{attribute 'GeneratedUsingTerminal: IODEVICETYPE_ETHERCATPROT'}
{attribute addProperty BoxType "IODEVICETYPE_ETHERCATPROT"}
{attribute addProperty Id "Beckhoff_BKxxxxBeckhoff_BKxxxx_735133AB0Beckhoff_CUxxxxBeckhoff_CUxxxx_E18DC8DB94Beckhoff_CXxxxxBeckhoff_CXxxxx_C55F0A74176TcTerminals210_EK1100_1TcTerminals210_EK1100_1_5C7783790TcTerminals210_EK1100_2TcTerminals210_EK1100_2_50C143310SyncUnitsSyncUnits_99E584AF18InputsInputs_25A0042B160OutputsOutputs_2397A10E106InfoDataInfoData_C76BEFB322"}
{attribute addProperty CRC "296101675"}
{attribute addProperty Size "576"}
TYPE EtherCAT_Master_BKCUCX_11A6272B :
STRUCT
	{attribute addProperty Name "Beckhoff_BKxxxx"}
	{attribute addProperty PreviousPort "EtherCAT_Master_BKCUCX : Master"}
	Beckhoff_BKxxxx : Beckhoff_BKxxxx_735133AB;
	{attribute addProperty Name "Beckhoff_CUxxxx"}
	{attribute addProperty PreviousPort "Beckhoff BKxxxx : C"}
	Beckhoff_CUxxxx : Beckhoff_CUxxxx_E18DC8DB;
	{attribute addProperty Name "Beckhoff_CXxxxx"}
	{attribute addProperty PreviousPort "Beckhoff CUxxxx : C"}
	Beckhoff_CXxxxx : Beckhoff_CXxxxx_C55F0A74;
	{attribute addProperty Name "TcTerminals210_EK1100_1"}
	{attribute addProperty PreviousPort "Beckhoff CXxxxx : C"}
	TcTerminals210_EK1100_1 : TcTerminals210_EK1100_1_5C778379;
	{attribute addProperty Name "TcTerminals210_EK1100_2"}
	{attribute addProperty PreviousPort "TcTerminals210_EK1100_1 : C"}
	TcTerminals210_EK1100_2 : TcTerminals210_EK1100_2_50C14331;
	{attribute addProperty Name "SyncUnits"}
	SyncUnits : SyncUnits_99E584AF;
	{attribute addProperty Name "Inputs"}
	Inputs : Inputs_25A0042B;
	{attribute addProperty Name "Outputs"}
	Outputs : Outputs_2397A10E;
	{attribute addProperty Name "InfoData"}
	InfoData : InfoData_C76BEFB3;
END_STRUCT
END_TYPE

(* stored: Version 1.2.0.0, ProductVersion 3.1.4024.9
   DUT EtherCAT_Master_BKCUCX_11A6272B: Id {93250250-dbae-4e0e-a4a5-ad824e1b5e2b} *)
